(* Schneider Machine Expert - Basic project Pueba robledo, file version 2.8.0.0 *)
(* ProjectInformations: Name=Nuevo proyecto *)

HARDWARE
  Cpu 0: TM221CE24T
  ModuleExtensionObject 0: TM3TI4/G
  EthernetConfiguration: NetworkName=M221, IpAllocationMode=FixedAddress, IpAddress=192.168.13.63, SubnetMask=255.255.255.0
  SerialLineConfiguration: Baud=Baud19200, Parity=ParityEven, DataBits=DataBits8, StopBits=StopBits1, PhysicalMedium=PhysicalMediumRs485, TransmissionMode=TransmissionModeModbusRtu, SlaveId=1, Addressing=SlaveAddressing
  MastTask: UsePeriodScanMode=false, PeriodScan=100
  FastTask: Period=255
  CpuBehavior: StartingMode=StartAsPreviousState, AutoSaveRamOnEeprom=true, WatchdogPeriod=250

SYMBOLS  (address, symbol, comment, settings)
  %IW1.0      [Type=Type_ThermocoupleJ, Scope=Scope_Celsius, Minimum=-2000, Maximum=10000]

POU Nuevo POU
  (* SectionNumber=1 *)

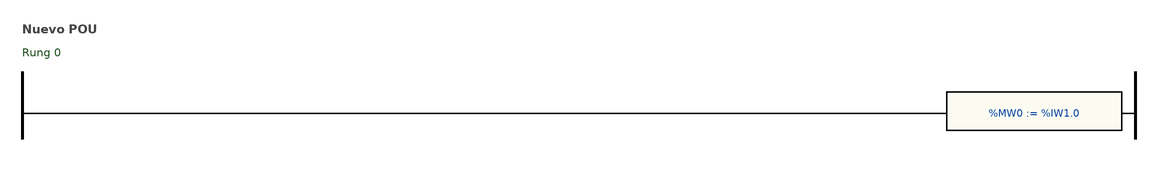

// Rung 0
  LD 1
  [ %MW0 := %IW1.0 ]
  // as ST:
  //   %MW0 := %IW1.0;
